{attribute 'qualified_only'}
VAR_GLOBAL
	NextfreeOrderID : INT;
	AktuellesStockwerk : INT;
END_VAR

(* stored: Version 1.1.0.1
   GVL OrderID_Counter: Id {2fe0a1d8-72a4-4413-84d3-4a8cd0c3527c} *)
